(* IEC 61131-3 sources: Std_PalletMover/Class/MQTTClient_Interface_Config, 1 file *)

(* ---- MQTTClient_Interface_Config.st ---- *)
(*!
<Class
	Name               = "MQTTClient_Interface_Config"
	Revision           = "1.1"
	RealtimeTask       = "false"
	CyclicTask         = "false"
	BackgroundTask     = "false"
	Sigmatek           = "true"
	OSInterface        = "false"
	HighPriority       = "false"
	Automatic          = "false"
	UpdateMode         = "Prescan"
	SharedCommandTable = "true"
	Objectsize         = "(844,120)"
	Comment            = "This class is used to configure the MQTTClient_Interface Class in conjunction with or as opposed to using the XML Configuration.&#13;&#10;The MQTTClient_Interface class first reads the XML configuration if present and the the configuration specified by this class.&#13;&#10;Most common settings are possible on this derivation of the MQTTClient_Interface_ConfigBase Class.">
	<Channels>
		<Server Name="CAFileString" Class="StringRAM" Visualized="true" Initialize="true" WriteProtected="false" Retentive="false" Comment="Object channel to the StringRAM object on which the CA Filename string is to be specified.&#13;&#10;&#13;&#10;The File should be placed in &quot;C:/LSLSYS/SSL/&quot; and the filename should be specified in the string:&#13;&#10;&#13;&#10;Example:&#13;&#10;Full path to the file is: &quot;C:/LSLSYS/SSL/myFile.cert&quot;&#13;&#10;String should contain: &quot;myFile.cert&quot;"/>
		<Server Name="CertFileString" Class="StringRAM" Visualized="true" Initialize="true" WriteProtected="false" Retentive="false" Comment="Object channel to the StringRAM object on which the Cert Filename string is to be specified.&#13;&#10;&#13;&#10;The File should be placed in &quot;C:/LSLSYS/SSL/&quot; and the filename should be specified in the string:&#13;&#10;&#13;&#10;Example:&#13;&#10;Full path to the file is: &quot;C:/LSLSYS/SSL/myFile.cert&quot;&#13;&#10;String should contain: &quot;myFile.cert&quot;"/>
		<Server Name="ClientIDString" Class="StringRAM" Visualized="true" Initialize="true" WriteProtected="false" Retentive="false" Comment="Object channel to the StringRAM object on which the ClientID string is to be specified.&#13;&#10;&#13;&#10;If not specified the XML Value / CPU Serial number is used."/>
		<Server Name="Exponential" Visualized="false" Initialize="true" DefValue="0" WriteProtected="false" Retentive="File" Comment="Whether the reconnection delay should increase exponentially should be specified on this server.&#13;&#10;0 = Linear Increase. (MinInterval must be &gt;= 1).&#13;&#10;1 = Exponential Increase. (MinInterval must be &gt;= 2).&#13;&#10;&#13;&#10;With MinInterval = 2 and MaxInterval = 30, Reconnection Intervals will be:&#13;&#10;0: 2,4,6,8,10,...,30,30,30,...&#13;&#10;1: 2,4,8,16,30,30,30,..."/>
		<Server Name="HostnameString" Class="StringRAM" Visualized="true" Initialize="true" WriteProtected="false" Retentive="false" Comment="Object channel to the StringRAM object on which the Hostname string is to be specified."/>
		<Server Name="KeepAlive" Visualized="false" Initialize="true" DefValue="60" WriteProtected="false" Retentive="File" Comment="KeepAlive time in seconds is to be specified on this server.&#13;&#10;&#13;&#10;Default = 60."/>
		<Server Name="KeyFilePassString" Class="StringRAM" Visualized="true" Initialize="true" WriteProtected="false" Retentive="false" Comment="Object channel to the StringRAM object on which the KeyFile Password string is to be specified."/>
		<Server Name="KeyFileString" Class="StringRAM" Visualized="true" Initialize="true" WriteProtected="false" Retentive="false" Comment="Object channel to the StringRAM object on which the Key Filename string is to be specified.&#13;&#10;&#13;&#10;The File should be placed in &quot;C:/LSLSYS/SSL/&quot; and the filename should be specified in the string:&#13;&#10;&#13;&#10;Example:&#13;&#10;Full path to the file is: &quot;C:/LSLSYS/SSL/myFile.cert&quot;&#13;&#10;String should contain: &quot;myFile.cert&quot;"/>
		<Server Name="MaxInflightMsgs" Visualized="false" Initialize="true" DefValue="20" WriteProtected="false" Retentive="File" Comment="Maximum number of inflight messages are to be specified on this server.&#13;&#10;In a standard application this value should not be changed.&#13;&#10;&#13;&#10;Default = 20."/>
		<Server Name="MaxInterval" Visualized="false" Initialize="true" DefValue="30" WriteProtected="false" Retentive="File" Comment="Maximum delay interval to be used for the reconnection procedure, should be specified in seconds.&#13;&#10;&#13;&#10;Default = 30."/>
		<Server Name="MinInterval" Visualized="false" Initialize="true" DefValue="2" WriteProtected="false" Retentive="File" Comment="Minimum delay interval to be used for the reconnection procedure, should be specified in seconds.&#13;&#10;&#13;&#10;Default = 2."/>
		<Server Name="PasswordString" Class="StringRAM" Visualized="true" Initialize="true" WriteProtected="false" Retentive="false" Comment="Object channel to the StringRAM object on which the Password string is to be specified."/>
		<Server Name="Port" Visualized="false" Initialize="true" DefValue="1883" WriteProtected="false" Retentive="File" Comment="Connection port number is to be specified on this server, defaults are:&#13;&#10;&#13;&#10;Non-Encrypted: 1833&#13;&#10;Encrypted (No Client Cert): 8883&#13;&#10;Encrypted (With Client Cert): 8884&#13;&#10;&#13;&#10;Default = 1883."/>
		<Server Name="SetAuthenticationParameters" Visualized="false" Initialize="true" DefValue="0" WriteProtected="false" Retentive="File" Comment="On this server the user must specify whether the Authentication Parameters are to be set or ignored during configuration, if ignored the default / XML configured values will be used by the MQTTClient_Interface instance.&#13;&#10;&#13;&#10;Default = 0."/>
		<Server Name="SetCAFile" Visualized="false" Initialize="true" DefValue="0" WriteProtected="false" Retentive="File" Comment="On this server the user must specify whether the TLS - CA File is to be specified or ignored during configuration, if ignored the default / XML configured value will be used by the MQTTClient_Interface instance.&#13;&#10;&#13;&#10;Default = 0."/>
		<Server Name="SetCertFile" Visualized="false" Initialize="true" DefValue="0" WriteProtected="false" Retentive="File" Comment="On this server the user must specify whether the TLS - Cert File is to be specified or ignored during configuration, if ignored the default / XML configured value will be used by the MQTTClient_Interface instance.&#13;&#10;&#13;&#10;Default = 0."/>
		<Server Name="SetClientID" Visualized="false" Initialize="true" DefValue="0" WriteProtected="false" Retentive="File" Comment="On this server the user must specify whether the ClientID is to be set or ignored during configuration, if ignored the default / XML configured value will be used by the MQTTClient_Interface instance.&#13;&#10;&#13;&#10;Default = 0."/>
		<Server Name="SetConnectionParameters" Visualized="false" Initialize="true" DefValue="0" WriteProtected="false" Retentive="File" Comment="On this server the user must specify whether the Connection Parameters are to be set or ignored during configuration, if ignored the default / XML configured values will be used by the MQTTClient_Interface instance.&#13;&#10;&#13;&#10;Default = 0."/>
		<Server Name="SetKeyFile" Visualized="false" Initialize="true" DefValue="0" WriteProtected="false" Retentive="File" Comment="On this server the user must specify whether the TLS - Key File is to be specified or ignored during configuration, if ignored the default / XML configured value will be used by the MQTTClient_Interface instance.&#13;&#10;&#13;&#10;Default = 0."/>
		<Server Name="SetKeyFilePass" Visualized="false" Initialize="true" DefValue="0" WriteProtected="false" Retentive="File" Comment="On this server the user must specify whether the TLS - Key File Password is to be specified or ignored during configuration, if ignored the default / XML configured value will be used by the MQTTClient_Interface instance.&#13;&#10;&#13;&#10;Default = 0."/>
		<Server Name="SetMaxInflightMsgs" Visualized="false" Initialize="true" DefValue="0" WriteProtected="false" Retentive="File" Comment="On this server the user must specify whether the Max Inflight Messages value is to be set or ignored during configuration, if ignored the default / XML configured value will be used by the MQTTClient_Interface instance.&#13;&#10;&#13;&#10;Default = 0."/>
		<Server Name="SetReconnectionParameters" Visualized="false" Initialize="true" DefValue="0" WriteProtected="false" Retentive="File" Comment="On this server the user must specify whether the Reconnection Parameters are to be set or ignored during configuration, if ignored the default / XML configured values will be used by the MQTTClient_Interface instance.&#13;&#10;&#13;&#10;Default = 0."/>
		<Server Name="SetWillParameters" Visualized="false" Initialize="true" DefValue="0" WriteProtected="false" Retentive="File" Comment="On this server the user must specify whether the Will Parameters are to be set or ignored during configuration, if ignored the default / XML configured values will be used by the MQTTClient_Interface instance.&#13;&#10;&#13;&#10;Default = 0."/>
		<Server Name="UsernameString" Class="StringRAM" Visualized="true" Initialize="true" WriteProtected="false" Retentive="false" Comment="Object channel to the StringRAM object on which the Username string is to be specified."/>
		<Server Name="WillQoS" Visualized="false" Initialize="true" DefValue="0" WriteProtected="false" Retentive="File" Comment="Quality of Service (QoS) to be used for the Will Message delivery.&#13;&#10;&#13;&#10;Possible Values = 0,1,2.&#13;&#10;Default = 0."/>
		<Server Name="WillRetained" Visualized="false" Initialize="true" WriteProtected="false" Retentive="File" Comment="Whether the Will Message is to be retained on the broker for new clients to receive when connecting after this will has been published.&#13;&#10;&#13;&#10;0 = Not Retained.&#13;&#10;1 = Retained.&#13;&#10;&#13;&#10;Default = 0."/>
		<Server Name="WillText" Class="StringRAM" Visualized="true" Initialize="true" WriteProtected="false" Retentive="false" Comment="Object channel to the StringRAM object on which the Will Text string is to be specified."/>
		<Server Name="WillTopic" Class="StringRAM" Visualized="true" Initialize="true" WriteProtected="false" Retentive="false" Comment="Object channel to the StringRAM object on which the Will Topic string is to be specified."/>
		<Client Name="CAFilePathStringObject" Required="true" Internal="true"/>
		<Client Name="CertFilePathStringObject" Required="true" Internal="true"/>
		<Client Name="ClientIDStringObject" Required="true" Internal="true"/>
		<Client Name="HostnameStringObject" Required="true" Internal="true"/>
		<Client Name="KeyFilePathStringObject" Required="true" Internal="true"/>
		<Client Name="PasswordStringObject" Required="true" Internal="true"/>
		<Client Name="SigCLib" Required="false" Internal="false" Comment="Object Channel to the SigCLib Client Interface, should not be connected by the user."/>
		<Client Name="TLSPasswordStringObject" Required="true" Internal="true"/>
		<Client Name="UsernameStringObject" Required="true" Internal="true"/>
		<Client Name="WillTextStringObject" Required="true" Internal="true"/>
		<Client Name="WillTopicStringObject" Required="true" Internal="true"/>
	</Channels>
	<Separators>
		<Servers>
			<SepChn Position="3"/>
			<SepChn Position="0"/>
			<SepChn Position="8"/>
			<SepChn Position="11"/>
			<SepChn Position="16"/>
			<SepChn Position="22"/>
			<SepChn Position="26"/>
		</Servers>
	</Separators>
	<Dependencies>
		<Files>
			<File Path=".\Class\MQTTClient_Interface_Config\MQTTClient_Interface_Config_de.pdf"/>
			<File Path=".\Class\MQTTClient_Interface_Config\MQTTClient_Interface_Config_en.pdf"/>
		</Files>
	</Dependencies>
	<RevDoku>
		<Owner Company="Sigmatek" Author="VelGer"/>
		<Dokumentation Revision="1.1" Date="2019-06-12" Author="VelGer" Company="Sigmatek" Description="Server Comments Corrected."/>
		<Dokumentation Revision="1.0" Date="2019-05-08" Author="VelGer" Company="Sigmatek" Description="Initial Creation."/>
	</RevDoku>
	<Network Name="MQTTClient_Interface_Config">
		<!-- List of Components in this network -->
		<Components>
			<Object
				Name       = "_base"
				Class      = "MQTTClient_Interface_ConfigBase"
				Position   = "(218,120)"
				Visualized = "false">
				<Channels>
					<Server Name="LoginOK"/>
					<Client Name="MQTTClient_Interface"/>
				</Channels>
			</Object>
			<Object
				Name       = "CAFilePathStringObject"
				Class      = "StringRAM"
				Position   = "(120,2070)"
				Visualized = "true"
				Remotely   = "true">
				<Channels>
					<Server Name="Data"/>
					<Client Name="SingleRealloc" Value="1"/>
					<Client Name="UseFile"/>
				</Channels>
			</Object>
			<Object
				Name       = "CertFilePathStringObject"
				Class      = "StringRAM"
				Position   = "(120,2340)"
				Visualized = "true"
				Remotely   = "true">
				<Channels>
					<Server Name="Data"/>
					<Client Name="SingleRealloc" Value="1"/>
					<Client Name="UseFile"/>
				</Channels>
			</Object>
			<Object
				Name       = "ClientIDStringObject"
				Class      = "StringRAM"
				Position   = "(120,420)"
				Visualized = "true"
				Remotely   = "true">
				<Channels>
					<Server Name="Data"/>
					<Client Name="SingleRealloc" Value="1"/>
					<Client Name="UseFile" Value="1"/>
				</Channels>
			</Object>
			<Object
				Name       = "HostnameStringObject"
				Class      = "StringRAM"
				Position   = "(120,720)"
				Visualized = "true"
				Remotely   = "true">
				<Channels>
					<Server Name="Data"/>
					<Client Name="SingleRealloc" Value="1"/>
					<Client Name="UseFile" Value="1"/>
				</Channels>
			</Object>
			<Object
				Name       = "KeyFilePathStringObject"
				Class      = "StringRAM"
				Position   = "(120,2610)"
				Visualized = "true"
				Remotely   = "true">
				<Channels>
					<Server Name="Data"/>
					<Client Name="SingleRealloc" Value="1"/>
					<Client Name="UseFile"/>
				</Channels>
			</Object>
			<Object
				Name       = "PasswordStringObject"
				Class      = "StringRAM"
				Position   = "(120,1800)"
				Visualized = "true"
				Remotely   = "true">
				<Channels>
					<Server Name="Data"/>
					<Client Name="SingleRealloc" Value="1"/>
					<Client Name="UseFile" Value="1"/>
				</Channels>
			</Object>
			<Object
				Name       = "TLSPasswordStringObject"
				Class      = "StringRAM"
				Position   = "(120,2880)"
				Visualized = "true"
				Remotely   = "true">
				<Channels>
					<Server Name="Data"/>
					<Client Name="SingleRealloc" Value="1"/>
					<Client Name="UseFile"/>
				</Channels>
			</Object>
			<Object
				Name       = "UsernameStringObject"
				Class      = "StringRAM"
				Position   = "(120,1530)"
				Visualized = "true"
				Remotely   = "true">
				<Channels>
					<Server Name="Data"/>
					<Client Name="SingleRealloc" Value="1"/>
					<Client Name="UseFile" Value="1"/>
				</Channels>
			</Object>
			<Object
				Name       = "WillTextStringObject"
				Class      = "StringRAM"
				Position   = "(120,1260)"
				Visualized = "true"
				Remotely   = "true">
				<Channels>
					<Server Name="Data"/>
					<Client Name="SingleRealloc" Value="1"/>
					<Client Name="UseFile" Value="1"/>
				</Channels>
			</Object>
			<Object
				Name       = "WillTopicStringObject"
				Class      = "StringRAM"
				Position   = "(120,990)"
				Visualized = "true"
				Remotely   = "true">
				<Channels>
					<Server Name="Data"/>
					<Client Name="SingleRealloc" Value="1"/>
					<Client Name="UseFile" Value="1"/>
				</Channels>
			</Object>
		</Components>
		<Comments>
			<Comment Position="(900,2130)" Size="(180,150)" Text="Use property window to enter text."/>
		</Comments>
		<!-- List of Connections in this network -->
		<Connections>
			<Connection Source="this.LoginOK" Destination="_base.LoginOK" Vertices="(1236,210),(518,210),"/>
			<Connection Source="_base.MQTTClient_Interface" Destination="this.MQTTClient_Interface" Vertices="(218,210),(38,210),"/>
			<Connection Source="this.ClientIDStringObject" Destination="ClientIDStringObject.Data"/>
			<Connection Source="this.ClientIDString" Destination="ClientIDStringObject.Data" Vertices="(1236,330),(660,330),(630,360),(630,480),(600,510),(706,510),"/>
			<Connection Source="this.HostnameStringObject" Destination="HostnameStringObject.Data"/>
			<Connection Source="this.HostnameString" Destination="HostnameStringObject.Data" Vertices="(1236,450),(720,450),(690,480),(690,780),(660,810),(706,810),"/>
			<Connection Source="this.WillTopicStringObject" Destination="WillTopicStringObject.Data"/>
			<Connection Source="this.WillTextStringObject" Destination="WillTextStringObject.Data"/>
			<Connection Source="this.WillTopic" Destination="WillTopicStringObject.Data" Vertices="(1236,1050),(630,1050),(600,1080),(706,1080),"/>
			<Connection Source="this.WillText" Destination="WillTextStringObject.Data" Vertices="(1236,1110),(660,1110),(630,1140),(630,1320),(600,1350),(706,1350),"/>
			<Connection Source="this.UsernameStringObject" Destination="UsernameStringObject.Data"/>
			<Connection Source="this.UsernameString" Destination="UsernameStringObject.Data" Vertices="(1236,1350),(660,1350),(630,1380),(630,1590),(600,1620),(706,1620),"/>
			<Connection Source="this.PasswordStringObject" Destination="PasswordStringObject.Data"/>
			<Connection Source="this.PasswordString" Destination="PasswordStringObject.Data" Vertices="(1236,1410),(690,1410),(660,1440),(660,1860),(630,1890),(706,1890),"/>
			<Connection Source="this.CAFilePathStringObject" Destination="CAFilePathStringObject.Data"/>
			<Connection Source="this.CertFilePathStringObject" Destination="CertFilePathStringObject.Data"/>
			<Connection Source="this.KeyFilePathStringObject" Destination="KeyFilePathStringObject.Data"/>
			<Connection Source="this.TLSPasswordStringObject" Destination="TLSPasswordStringObject.Data"/>
			<Connection Source="this.CAFileString" Destination="CAFilePathStringObject.Data" Vertices="(1236,1530),(720,1530),(690,1560),(690,2130),(660,2160),(706,2160),"/>
			<Connection Source="this.CertFileString" Destination="CertFilePathStringObject.Data" Vertices="(1236,1650),(750,1650),(720,1680),(720,2400),(690,2430),(706,2430),"/>
			<Connection Source="this.KeyFileString" Destination="KeyFilePathStringObject.Data" Vertices="(1236,1770),(780,1770),(750,1800),(750,2670),(720,2700),(706,2700),"/>
			<Connection Source="this.KeyFilePassString" Destination="TLSPasswordStringObject.Data" Vertices="(1236,1890),(810,1890),(780,1920),(780,2940),(750,2970),(706,2970),"/>
		</Connections>
		<!-- Headerfiles -->
		<Options>
		</Options>
	</Network>
</Class>
*)
#pragma using MQTTClient_Interface_ConfigBase

MQTTClient_Interface_Config : CLASS
: MQTTClient_Interface_ConfigBase
  //Servers:
	SetClientID 	: SvrCh_DINT;
	ClientIDString 	: SvrChCmd_UDINT;
	SetConnectionParameters 	: SvrCh_DINT;
	HostnameString 	: SvrChCmd_UDINT;
	KeepAlive 	: SvrCh_DINT;
	Port 	: SvrCh_DINT;
	SetMaxInflightMsgs 	: SvrCh_DINT;
	MaxInflightMsgs 	: SvrCh_DINT;
	SetReconnectionParameters 	: SvrCh_DINT;
	MinInterval 	: SvrCh_DINT;
	MaxInterval 	: SvrCh_DINT;
	Exponential 	: SvrCh_DINT;
	SetWillParameters 	: SvrCh_DINT;
	WillTopic 	: SvrChCmd_UDINT;
	WillText 	: SvrChCmd_UDINT;
	WillQoS 	: SvrCh_DINT;
	WillRetained 	: SvrCh_DINT;
	SetAuthenticationParameters 	: SvrCh_DINT;
	UsernameString 	: SvrChCmd_UDINT;
	PasswordString 	: SvrChCmd_UDINT;
	SetCAFile 	: SvrCh_DINT;
	CAFileString 	: SvrChCmd_UDINT;
	SetCertFile 	: SvrCh_DINT;
	CertFileString 	: SvrChCmd_UDINT;
	SetKeyFile 	: SvrCh_DINT;
	KeyFileString 	: SvrChCmd_UDINT;
	SetKeyFilePass 	: SvrCh_DINT;
	KeyFilePassString 	: SvrChCmd_UDINT;
  //Clients:
	SigCLib 	: CltChCmd_SigCLib;
	ClientIDStringObject 	: CltChCmd_StringRAM;
	HostnameStringObject 	: CltChCmd_StringRAM;
	WillTopicStringObject 	: CltChCmd_StringRAM;
	WillTextStringObject 	: CltChCmd_StringRAM;
	UsernameStringObject 	: CltChCmd_StringRAM;
	PasswordStringObject 	: CltChCmd_StringRAM;
	TLSPasswordStringObject 	: CltChCmd_StringRAM;
	CAFilePathStringObject 	: CltChCmd_StringRAM;
	CertFilePathStringObject 	: CltChCmd_StringRAM;
	KeyFilePathStringObject 	: CltChCmd_StringRAM;
  //Variables:
		aClientID : ARRAY [0..MQTT_PROT_MAX_CLIENTID_NAME_LEN] OF UINT;

		aHostname : ARRAY [0..MQTTCLIENT_HOSTNAME_MAX_LEN] OF UINT;

		iPort 	: INT;
		iKeepAlive 	: INT;
		iMaxInflight 	: INT;
		aUsername : ARRAY [0..MQTTCLIENTINTERFACE_CONNECT_USERNAME_MAX_LEN] OF UINT;

		aPassword : ARRAY [0..MQTTCLIENTINTERFACE_CONNECT_PASSWORD_MAX_LEN] OF UINT;

		aWillTopic : ARRAY [0..MQTTCLIENTINTERFACE_WILL_TOPIC_MAX_LEN] OF UINT;

		aWillMessage : ARRAY [0..MQTTCLIENTINTERFACE_WILL_PAYLOAD_MAX_LEN] OF CHAR;

		iWillQoS 	: INT;
		bWillRetain 	: BOOL;
		iReconnMin 	: INT;
		iReconnMax 	: INT;
		bReconnExp 	: BOOL;
		aCAFile : ARRAY [0..MQTTCLIENTINTERFACE_TLS_CAFILE_MAX_LEN] OF CHAR;

		aCertFile : ARRAY [0..MQTTCLIENTINTERFACE_TLS_CERTFILE_MAX_LEN] OF CHAR;

		aKeyFile : ARRAY [0..MQTTCLIENTINTERFACE_TLS_KEYFILE_MAX_LEN] OF CHAR;

		aTLSPassword : ARRAY [0..MQTTCLIENTINTERFACE_TLS_PASSWORD_MAX_LEN] OF CHAR;

  //Functions:

	FUNCTION VIRTUAL GLOBAL ClientID
		VAR_OUTPUT
			Data 	: t_s_ClientID;
		END_VAR;

	FUNCTION VIRTUAL GLOBAL ConnectionParameters
		VAR_OUTPUT
			Data 	: t_s_ConnectionParameters;
		END_VAR;

	FUNCTION VIRTUAL GLOBAL MaxInflightMessages
		VAR_OUTPUT
			Data 	: t_s_MaxInflightMessages;
		END_VAR;

	FUNCTION VIRTUAL GLOBAL ReconnectionParameters
		VAR_OUTPUT
			Data 	: t_s_ReconnectionParameters;
		END_VAR;

	FUNCTION VIRTUAL GLOBAL Will
		VAR_OUTPUT
			Data 	: t_s_Will;
		END_VAR;

	FUNCTION VIRTUAL GLOBAL AuthenticationParameters
		VAR_OUTPUT
			Data 	: t_s_Authentication;
		END_VAR;

	FUNCTION VIRTUAL GLOBAL TLS
		VAR_OUTPUT
			Data 	: t_s_TLS;
		END_VAR;

	FUNCTION VIRTUAL GLOBAL ClientIDString::Read
		VAR_OUTPUT
			output (EAX) 	: UDINT;
		END_VAR;

	FUNCTION VIRTUAL GLOBAL ClientIDString::Write
		VAR_INPUT
			input (EAX) 	: UDINT;
		END_VAR
		VAR_OUTPUT
			result (EAX) 	: UDINT;
		END_VAR;

	FUNCTION VIRTUAL GLOBAL HostnameString::Read
		VAR_OUTPUT
			output (EAX) 	: UDINT;
		END_VAR;

	FUNCTION VIRTUAL GLOBAL HostnameString::Write
		VAR_INPUT
			input (EAX) 	: UDINT;
		END_VAR
		VAR_OUTPUT
			result (EAX) 	: UDINT;
		END_VAR;

	FUNCTION VIRTUAL GLOBAL WillTopic::Read
		VAR_OUTPUT
			output (EAX) 	: UDINT;
		END_VAR;

	FUNCTION VIRTUAL GLOBAL WillTopic::Write
		VAR_INPUT
			input (EAX) 	: UDINT;
		END_VAR
		VAR_OUTPUT
			result (EAX) 	: UDINT;
		END_VAR;

	FUNCTION VIRTUAL GLOBAL WillText::Read
		VAR_OUTPUT
			output (EAX) 	: UDINT;
		END_VAR;

	FUNCTION VIRTUAL GLOBAL WillText::Write
		VAR_INPUT
			input (EAX) 	: UDINT;
		END_VAR
		VAR_OUTPUT
			result (EAX) 	: UDINT;
		END_VAR;

	FUNCTION VIRTUAL GLOBAL UsernameString::Read
		VAR_OUTPUT
			output (EAX) 	: UDINT;
		END_VAR;

	FUNCTION VIRTUAL GLOBAL UsernameString::Write
		VAR_INPUT
			input (EAX) 	: UDINT;
		END_VAR
		VAR_OUTPUT
			result (EAX) 	: UDINT;
		END_VAR;

	FUNCTION VIRTUAL GLOBAL PasswordString::Read
		VAR_OUTPUT
			output (EAX) 	: UDINT;
		END_VAR;

	FUNCTION VIRTUAL GLOBAL PasswordString::Write
		VAR_INPUT
			input (EAX) 	: UDINT;
		END_VAR
		VAR_OUTPUT
			result (EAX) 	: UDINT;
		END_VAR;

	FUNCTION VIRTUAL GLOBAL CAFileString::Read
		VAR_OUTPUT
			output (EAX) 	: UDINT;
		END_VAR;

	FUNCTION VIRTUAL GLOBAL CAFileString::Write
		VAR_INPUT
			input (EAX) 	: UDINT;
		END_VAR
		VAR_OUTPUT
			result (EAX) 	: UDINT;
		END_VAR;

	FUNCTION VIRTUAL GLOBAL CertFileString::Read
		VAR_OUTPUT
			output (EAX) 	: UDINT;
		END_VAR;

	FUNCTION VIRTUAL GLOBAL CertFileString::Write
		VAR_INPUT
			input (EAX) 	: UDINT;
		END_VAR
		VAR_OUTPUT
			result (EAX) 	: UDINT;
		END_VAR;

	FUNCTION VIRTUAL GLOBAL KeyFileString::Read
		VAR_OUTPUT
			output (EAX) 	: UDINT;
		END_VAR;

	FUNCTION VIRTUAL GLOBAL KeyFileString::Write
		VAR_INPUT
			input (EAX) 	: UDINT;
		END_VAR
		VAR_OUTPUT
			result (EAX) 	: UDINT;
		END_VAR;

	FUNCTION VIRTUAL GLOBAL KeyFilePassString::Read
		VAR_OUTPUT
			output (EAX) 	: UDINT;
		END_VAR;

	FUNCTION VIRTUAL GLOBAL KeyFilePassString::Write
		VAR_INPUT
			input (EAX) 	: UDINT;
		END_VAR
		VAR_OUTPUT
			result (EAX) 	: UDINT;
		END_VAR;
  //Tables:
	FUNCTION @STD
		VAR_OUTPUT
			ret_code	: CONFSTATES;
		END_VAR;
	FUNCTION GLOBAL TAB @CT_;
END_CLASS;

#pragma using StringRAM
#pragma usingLtd SigCLib

FUNCTION VIRTUAL GLOBAL MQTTClient_Interface_Config::ClientID
	VAR_OUTPUT
		Data 	: t_s_ClientID;
	END_VAR

  //Set the ClientID if active, else return defaults
  if SetClientID = 1 then

    //==================================CLIENT ID
    //Clear out ClientID
    SigCLib.MemSet(dst  :=  #aClientID,
                   c    :=  0x00,
                   len  :=  sizeof(aClientID));

    //Read the string object into the local buffer
    ClientIDStringObject.ToUniCode();
    ClientIDStringObject.TxtGet(pdst    :=  #aClientID[0],
                                dstsize :=  sizeof(aClientID));

    //Set the Return Pointer
    Data.ClientID := #aClientID[0];

  else

    Data := MQTTClient_Interface_ConfigBase::ClientID();

  end_if;

END_FUNCTION

FUNCTION VIRTUAL GLOBAL MQTTClient_Interface_Config::ConnectionParameters
	VAR_OUTPUT
		Data 	: t_s_ConnectionParameters;
	END_VAR

  //Set the Connection Parameters if active, else return defaults.
  if SetConnectionParameters = 1 then

    //==================================HOSTNAME
    //Clear out Hostname
    SigCLib.MemSet(dst  :=  #aHostname,
                   c    :=  0x00,
                   len  :=  sizeof(aHostname));

    //Read the string object into the local buffer
    HostnameStringObject.ToUniCode();
    HostnameStringObject.TxtGet(pdst    :=  #aHostname[0],
                                dstsize :=  sizeof(aHostname));

    //Set the Return Pointer
    Data.hostname := #aHostname[0];

    //==================================PORT

    Data.keepalive := to_int(KeepAlive);

    //==================================KEEPALIVE

    Data.port := to_int(Port);

  else

    Data := MQTTClient_Interface_ConfigBase::ConnectionParameters();

  end_if;

END_FUNCTION

FUNCTION VIRTUAL GLOBAL MQTTClient_Interface_Config::ClientIDString::Read
	VAR_OUTPUT
		output (EAX) 	: UDINT;
	END_VAR

	ClientIDString := ClientIDStringObject.Data.Read();
	output := ClientIDString;

END_FUNCTION

FUNCTION VIRTUAL GLOBAL MQTTClient_Interface_Config::ClientIDString::Write
	VAR_INPUT
		input (EAX) 	: UDINT;
	END_VAR
	VAR_OUTPUT
		result (EAX) 	: UDINT;
	END_VAR

	ClientIDString := input;
	result := (ClientIDStringObject.Data.Write(ClientIDString))$UDINT;

END_FUNCTION

FUNCTION VIRTUAL GLOBAL MQTTClient_Interface_Config::HostnameString::Read
	VAR_OUTPUT
		output (EAX) 	: UDINT;
	END_VAR

	HostnameString := HostnameStringObject.Data.Read();
	output := HostnameString;

END_FUNCTION

FUNCTION VIRTUAL GLOBAL MQTTClient_Interface_Config::HostnameString::Write
	VAR_INPUT
		input (EAX) 	: UDINT;
	END_VAR
	VAR_OUTPUT
		result (EAX) 	: UDINT;
	END_VAR

	HostnameString := input;
	result := (HostnameStringObject.Data.Write(HostnameString))$UDINT;

END_FUNCTION

FUNCTION VIRTUAL GLOBAL MQTTClient_Interface_Config::MaxInflightMessages
	VAR_OUTPUT
		Data 	: t_s_MaxInflightMessages;
	END_VAR

  //Set the Max Inflight Messages if active, else return defaults.
  if SetMaxInflightMsgs = 1 then

    Data.max_inflight_messages := to_int(MaxInflightMsgs);

  else

    Data := MQTTClient_Interface_ConfigBase::MaxInflightMessages();

  end_if;

END_FUNCTION

FUNCTION VIRTUAL GLOBAL MQTTClient_Interface_Config::ReconnectionParameters
	VAR_OUTPUT
		Data 	: t_s_ReconnectionParameters;
	END_VAR

  //Set the Reconnection paramters if active, else return defaults.
  if SetReconnectionParameters = 1 then

    Data.min_interval       := to_int(MinInterval);
    Data.max_interval       := to_int(MaxInterval);
    Data.exponential_scale  := to_bool(Exponential);

  else

    Data := MQTTClient_Interface_ConfigBase::Reconnectionparameters();

  end_if;

END_FUNCTION

FUNCTION VIRTUAL GLOBAL MQTTClient_Interface_Config::WillTopic::Read
	VAR_OUTPUT
		output (EAX) 	: UDINT;
	END_VAR

	WillTopic := WillTopicStringObject.Data.Read();
	output := WillTopic;

END_FUNCTION

FUNCTION VIRTUAL GLOBAL MQTTClient_Interface_Config::WillTopic::Write
	VAR_INPUT
		input (EAX) 	: UDINT;
	END_VAR
	VAR_OUTPUT
		result (EAX) 	: UDINT;
	END_VAR

	WillTopic := input;
	result := (WillTopicStringObject.Data.Write(WillTopic))$UDINT;

END_FUNCTION

FUNCTION VIRTUAL GLOBAL MQTTClient_Interface_Config::WillText::Read
	VAR_OUTPUT
		output (EAX) 	: UDINT;
	END_VAR

	WillText := WillTextStringObject.Data.Read();
	output := WillText;

END_FUNCTION

FUNCTION VIRTUAL GLOBAL MQTTClient_Interface_Config::WillText::Write
	VAR_INPUT
		input (EAX) 	: UDINT;
	END_VAR
	VAR_OUTPUT
		result (EAX) 	: UDINT;
	END_VAR

	WillText := input;
	result := (WillTextStringObject.Data.Write(WillText))$UDINT;

END_FUNCTION

FUNCTION VIRTUAL GLOBAL MQTTClient_Interface_Config::Will
	VAR_OUTPUT
		Data 	: t_s_Will;
	END_VAR

  //Set the Will paramters if active, else return defaults.
  if SetWillParameters = 1 then

    //==================================TOPIC
    //Clear out Topic
    SigCLib.MemSet(dst  :=  #aWillTopic,
                   c    :=  0x00,
                   len  :=  sizeof(aWillTopic));

    //Read the string object into the local buffer
    WillTopicStringObject.ToUniCode();
    WillTopicStringObject.TxtGet(pdst    :=  #aWillTopic[0],
                                 dstsize :=  sizeof(aWillTopic));

    //Set the Return Pointer
    Data.topic := #aWillTopic[0];

    //==================================PAYLOAD
    //Clear out Payload
    SigCLib.MemSet(dst  :=  #aWillMessage,
                   c    :=  0x00,
                   len  :=  sizeof(aWillMessage));

    //Read the string object into the local buffer
    WillTextStringObject.TxtGet(pdst    :=  #aWillMessage[0],
                                dstsize :=  sizeof(aWillMessage));

    //Set the Return Pointer
    Data.payloadtext := #aWillMessage[0];

    //==================================QoS

    Data.qos := to_int(WillQoS);

    //==================================Retain

    Data.bRetain := to_bool(WillRetained);

  else

    Data := MQTTClient_Interface_ConfigBase::Will();

  end_if;

END_FUNCTION

FUNCTION VIRTUAL GLOBAL MQTTClient_Interface_Config::AuthenticationParameters
	VAR_OUTPUT
		Data 	: t_s_Authentication;
	END_VAR

  //Set the Authentication parameters if active, else return defaults.
  if SetAuthenticationParameters = 1 then

    //==================================USERNAME
    //Clear out Topic
    SigCLib.MemSet(dst  :=  #aUsername,
                   c    :=  0x00,
                   len  :=  sizeof(aUsername));

    //Read the string object into the local buffer
    UsernameStringObject.ToUniCode();
    UsernameStringObject.TxtGet(pdst    :=  #aUsername[0],
                                dstsize :=  sizeof(aUsername));

    //Set the Return Pointer
    Data.username := #aUsername[0];

    //==================================PASSWORD
    //Clear out Password
    SigCLib.MemSet(dst  :=  #aPassword,
                   c    :=  0x00,
                   len  :=  sizeof(aPassword));

    //Read the string object into the local buffer
    PasswordStringObject.ToUniCode();
    PasswordStringObject.TxtGet(pdst    :=  #aPassword[0],
                                dstsize :=  sizeof(aPassword));

    //Set the Return Pointer
    Data.password := #aPassword[0];

  else

    Data := MQTTClient_Interface_ConfigBase::AuthenticationParameters();

  end_if;

END_FUNCTION

FUNCTION VIRTUAL GLOBAL MQTTClient_Interface_Config::UsernameString::Read
	VAR_OUTPUT
		output (EAX) 	: UDINT;
	END_VAR

	UsernameString := UsernameStringObject.Data.Read();
	output := UsernameString;

END_FUNCTION

FUNCTION VIRTUAL GLOBAL MQTTClient_Interface_Config::UsernameString::Write
	VAR_INPUT
		input (EAX) 	: UDINT;
	END_VAR
	VAR_OUTPUT
		result (EAX) 	: UDINT;
	END_VAR

	UsernameString := input;
	result := (UsernameStringObject.Data.Write(UsernameString))$UDINT;

END_FUNCTION

FUNCTION VIRTUAL GLOBAL MQTTClient_Interface_Config::PasswordString::Read
	VAR_OUTPUT
		output (EAX) 	: UDINT;
	END_VAR

	PasswordString := PasswordStringObject.Data.Read();
	output := PasswordString;

END_FUNCTION

FUNCTION VIRTUAL GLOBAL MQTTClient_Interface_Config::PasswordString::Write
	VAR_INPUT
		input (EAX) 	: UDINT;
	END_VAR
	VAR_OUTPUT
		result (EAX) 	: UDINT;
	END_VAR

	PasswordString := input;
	result := (PasswordStringObject.Data.Write(PasswordString))$UDINT;

END_FUNCTION

FUNCTION VIRTUAL GLOBAL MQTTClient_Interface_Config::TLS
	VAR_OUTPUT
		Data 	: t_s_TLS;
	END_VAR

  //Set the TLS parameters if active, else return defaults.
  if SetCAFile      = 1 |
     SetCertFile    = 1 |
     SetKeyFile     = 1 |
     SetKeyFilePass = 1 then

    //Clear out pointers
    Data.cafile   := NIL;
    Data.certfile := NIL;
    Data.keyfile  := NIL;
    Data.pw       := NIL;

    //If the CAFile must be used, set the value
    if SetCAFile = 1 then

      SigCLib.MemSet( dst :=  #aCAFile,
                      c   :=  0x00,
                      len :=  sizeof(aCAFile));

      CAFilePathStringObject.TxtGet(pdst    :=  #aCAFile[0],
                                    dstsize :=  sizeof(aCAFile));

      Data.cafile := #aCAFile[0];

    end_if;

    //If the CertFile must be used, set the value
    if SetCertFile = 1 then

      SigCLib.MemSet( dst :=  #aCertFile,
                      c   :=  0x00,
                      len :=  sizeof(aCertFile));

      CertFilePathStringObject.TxtGet(pdst    :=  #aCertFile[0],
                                      dstsize :=  sizeof(aCertFile));

      Data.certfile := #aCertFile[0];

    end_if;

    //If the KeyFile must be used, set the value
    if SetKeyFile = 1 then

      SigCLib.MemSet( dst :=  #aKeyFile,
                      c   :=  0x00,
                      len :=  sizeof(aKeyFile));

      KeyFilePathStringObject.TxtGet( pdst    :=  #aKeyFile[0],
                                      dstsize :=  sizeof(aKeyFile));

      Data.keyfile := #aKeyFile[0];

    end_if;

    //If the Password must be used, set the value
    if SetKeyFilePass = 1 then

      SigCLib.MemSet( dst :=  #aTLSPassword,
                      c   :=  0x00,
                      len :=  sizeof(aTLSPassword));

      TLSPasswordStringObject.TxtGet( pdst    :=  #aTLSPassword[0],
                                      dstsize :=  sizeof(aTLSPassword));

      Data.pw := #aTLSPassword[0];

    end_if;

  else

    Data := MQTTClient_Interface_ConfigBase::TLS();

  end_if;

END_FUNCTION

FUNCTION VIRTUAL GLOBAL MQTTClient_Interface_Config::CAFileString::Read
	VAR_OUTPUT
		output (EAX) 	: UDINT;
	END_VAR

	CAFileString := CAFilePathStringObject.Data.Read();
	output := CAFileString;

END_FUNCTION

FUNCTION VIRTUAL GLOBAL MQTTClient_Interface_Config::CAFileString::Write
	VAR_INPUT
		input (EAX) 	: UDINT;
	END_VAR
	VAR_OUTPUT
		result (EAX) 	: UDINT;
	END_VAR

	CAFileString := input;
	result := (CAFilePathStringObject.Data.Write(CAFileString))$UDINT;

END_FUNCTION

FUNCTION VIRTUAL GLOBAL MQTTClient_Interface_Config::CertFileString::Read
	VAR_OUTPUT
		output (EAX) 	: UDINT;
	END_VAR

	CertFileString := CertFilePathStringObject.Data.Read();
	output := CertFileString;

END_FUNCTION

FUNCTION VIRTUAL GLOBAL MQTTClient_Interface_Config::CertFileString::Write
	VAR_INPUT
		input (EAX) 	: UDINT;
	END_VAR
	VAR_OUTPUT
		result (EAX) 	: UDINT;
	END_VAR

	CertFileString := input;
	result := (CertFilePathStringObject.Data.Write(CertFileString))$UDINT;

END_FUNCTION

FUNCTION VIRTUAL GLOBAL MQTTClient_Interface_Config::KeyFileString::Read
	VAR_OUTPUT
		output (EAX) 	: UDINT;
	END_VAR

	KeyFileString := KeyFilePathStringObject.Data.Read();
	output := KeyFileString;

END_FUNCTION

FUNCTION VIRTUAL GLOBAL MQTTClient_Interface_Config::KeyFileString::Write
	VAR_INPUT
		input (EAX) 	: UDINT;
	END_VAR
	VAR_OUTPUT
		result (EAX) 	: UDINT;
	END_VAR

	KeyFileString := input;
	result := (KeyFilePathStringObject.Data.Write(KeyFileString))$UDINT;

END_FUNCTION

FUNCTION VIRTUAL GLOBAL MQTTClient_Interface_Config::KeyFilePassString::Read
	VAR_OUTPUT
		output (EAX) 	: UDINT;
	END_VAR

	KeyFilePassString := TLSPasswordStringObject.Data.Read();
	output := KeyFilePassString;

END_FUNCTION

FUNCTION VIRTUAL GLOBAL MQTTClient_Interface_Config::KeyFilePassString::Write
	VAR_INPUT
		input (EAX) 	: UDINT;
	END_VAR
	VAR_OUTPUT
		result (EAX) 	: UDINT;
	END_VAR

	KeyFilePassString := input;
	result := (TLSPasswordStringObject.Data.Write(KeyFilePassString))$UDINT;

END_FUNCTION
